FUNCTION_BLOCK FB_Picker_1 EXTENDS FB_Picker

SUPER^(); 


_M_Picker_PosY_VISU(); //Compute Y position of Picker_1 to display on VISU

METHOD PRIVATE _M_Picker_PosY_VISU : BOOL
VAR_INPUT
END_VAR
IF TargetBuffer_Is_1 AND ((State = E_PickerFixedState.InPlacedPos) OR  (State = E_PickerFixedState.PartPlaced)) THEN 
	IF (TargetPosition_Buffer = 1 ) OR (TargetPosition_Buffer = 7 ) THEN 
		Picker_PosY_VISU_Sim := 2238 -530;
	ELSIF (TargetPosition_Buffer = 2 ) OR (TargetPosition_Buffer = 8) THEN	
		Picker_PosY_VISU_Sim := 2238 -477;
	ELSIF (TargetPosition_Buffer = 3 ) OR (TargetPosition_Buffer = 9) THEN	
		Picker_PosY_VISU_Sim := 2238 -411;
	ELSIF (TargetPosition_Buffer = 4 ) OR (TargetPosition_Buffer = 10) THEN	
		Picker_PosY_VISU_Sim := 2238 -329;
	ELSIF (TargetPosition_Buffer = 5 ) OR (TargetPosition_Buffer = 11) THEN	
		Picker_PosY_VISU_Sim := 2238 -265;
	ELSIF (TargetPosition_Buffer = 6 ) OR (TargetPosition_Buffer = 12) THEN	
		Picker_PosY_VISU_Sim := 2238 -199;
	END_IF
	
ELSIF TargetBuffer_Is_2 AND ((State = E_PickerFixedState.InPlacedPos) OR  (State = E_PickerFixedState.PartPlaced)) THEN 
	IF (TargetPosition_Buffer = 1 ) OR (TargetPosition_Buffer = 7 ) THEN 
		Picker_PosY_VISU_Sim := 2238 - 1181;
	ELSIF (TargetPosition_Buffer = 2 ) OR (TargetPosition_Buffer = 8) THEN	
		Picker_PosY_VISU_Sim := 2238 - 1101;
	ELSIF (TargetPosition_Buffer = 3 ) OR (TargetPosition_Buffer = 9) THEN	
		Picker_PosY_VISU_Sim := 2238 - 1033;
	ELSIF (TargetPosition_Buffer = 4 ) OR (TargetPosition_Buffer = 10) THEN	
		Picker_PosY_VISU_Sim := 2238 - 959;
	ELSIF (TargetPosition_Buffer = 5 ) OR (TargetPosition_Buffer = 11) THEN	
		Picker_PosY_VISU_Sim := 2238 - 884;
	ELSIF (TargetPosition_Buffer = 6 ) OR (TargetPosition_Buffer = 12) THEN	
		Picker_PosY_VISU_Sim := 2238 - 822;
	END_IF

ELSIF (State = E_PickerFixedState.InPickedPos) OR  (State = E_PickerFixedState.PartPicked) THEN 
	Picker_PosY_VISU_Sim := 2238;
END_IF

//Picker_PosY_VISU_Sim := 2238;
//TargetPosition_Buffer
END_METHOD

METHOD M_IdleState : BOOL
VAR_INPUT
END_VAR

IF Disable_Picker THEN 
	State := E_PickerFixedState.Idle;
END_IF
END_METHOD

METHOD M_MoveToPickPos : BOOL
VAR_INPUT
END_VAR

Sim_Time(IN := TRUE, PT := T#1S);

IF Sim_Time.Q THEN       //We assume in 1 seconds we go to Pick position; CassettePos for Mover1, BufferPos for Mover2
	Sim_Time(IN := FALSE);
	State := E_PickerFixedState.InPickedPos;
END_IF
END_METHOD

METHOD M_MoveToPlacePos : BOOL
VAR_INPUT
	Buffer_1_InUse : BOOL; //TRUE If Buffer_1 is Used, FALSE if Buffer_2 is Used by the Picker
	Buffer_Pos : UINT;     // Dictates the Buffer Slot the place handover takes place
END_VAR
//If Picker_1 then PlaceToCarrier; if  Picker_2  PlaceToBuffer
//State := E_MoverTransitionState.Placing;


Sim_Time(IN := TRUE, PT := T#1S);

IF Sim_Time.Q THEN   //We assume in 1 seconds we go to Pick position; BufferPos for Mover1, CarrierPos for Mover2
	Sim_Time(IN := FALSE);
	State := E_PickerFixedState.InPlacedPos;
END_IF
END_METHOD

END_FUNCTION_BLOCK

(* stored: Version 1.1.0.1, ProductVersion 3.1.4024.12
   POU FB_Picker_1: Id {91297915-e066-40a2-a7f5-28d2930e8691}, SpecialFunc None
   Folder Methods: Id {ad9e9f44-8bd6-4393-81e1-87f2a6721565}
   Folder Private: Id {e5992217-f556-464c-b2df-a3a8d2f86323}
   Folder Public: Id {b45d30c4-d547-4a6d-b37e-7c0dc8c418e9}
   Method _M_Picker_PosY_VISU: Id {53e67097-0526-427d-a395-65e4e302d4a4}
   Method M_IdleState: Id {21afa249-8f81-49d8-a84e-c6946593c4c5}
   Method M_MoveToPickPos: Id {f64fc3ca-7148-49e5-9864-e4dee441f6e8}
   Method M_MoveToPlacePos: Id {2e459992-cfe1-4ff9-ad47-0e875ce65f90} *)
